FUNCTION_BLOCK fbDataExchangePIM
VAR_IN_OUT
	stMachineDataPIM : stPimMachineData;
END_VAR
VAR_INPUT
	//All purpose data
	sIpAdress 						: STRING(15);				// Ip Adress of machine
	iPort							: UINT;						// Port of the machine
	iUnitId							: BYTE;						// Id of Slave
	tCommunicationTimeOut			: TIME;						// Time until error 
	iCommunicationPerformEvery		: INT;						// Perform data exchange every ms
	bEnableCommunication			: BOOL;						// Enable communication
	//Byte purpose data
	wRegistersReadQuantity			: WORD;						// Amount of data do read
	wRegistersWriteQuantity			: WORD;						// Amount of data do read
	iRegisterReadStartAdress		: UINT;						// First adress of read registers data
	iRegisterWriteStartAdress		: UINT;						// First adress of write registers data
	iMaxCommunicationCycleTime		: INT;						//Maximum cycles to perform communication without error
END_VAR
VAR_OUTPUT
	bCommunicationError				: BOOL;						//Block state informaing about communication error
	iCommunicationErrorCode			: UDINT;					//Block state informaing about communication error
	bCommunicationBlockCycleExtended: BOOL;						//Communication Cycle extened
	iCommunicationCycleTime			: INT;						//
END_VAR

VAR
	iCommunicationStep 				: INT;	
	iCycleCalc						: INT;
	iLastCycleTimeClear				: TON;
	fbModbusTCP 					: FB_MBReadWriteRegs;
	arRegisterReadArray				: ARRAY[0..29] OF INT;
	arRegisterWriteArray			: ARRAY[0..29] OF INT;
	iHistoryError					: INT;
	arModbusErrorHist				: ARRAY[0..100] OF UDINT;
	iLasthistory					: INT;
END_VAR

//--------------------------------------------------------------------------------------------------
//Communication monitor
IF iCycleCalc > iMaxCommunicationCycleTime THEN
	bCommunicationError := TRUE;
	bCommunicationBlockCycleExtended := TRUE;
ELSIF fbModbusTCP.bError THEN
	bCommunicationError := TRUE;
	bCommunicationBlockCycleExtended := FALSE;
ELSE
	bCommunicationError := FALSE;
	bCommunicationBlockCycleExtended := FALSE;
END_IF
iCommunicationErrorCode := fbModbusTCP.nErrId;
IF iCycleCalc > iCommunicationCycleTime	  THEN
	iCommunicationCycleTime	:= iCycleCalc;
END_IF
iLastCycleTimeClear(IN:=TRUE,PT:=T#100MS);
IF iLastCycleTimeClear.Q THEN
	iCommunicationCycleTime := 0;
	iLastCycleTimeClear(IN:=FALSE);
END_IF
//--------------------------------------------------------------------------------------------------
//Statistic
//--------------------------------------------------------------------------------------------------
//Cycle counter
IF bEnableCommunication THEN
	iCycleCalc := iCycleCalc +1;
ELSE
	iCycleCalc := 0;
END_IF

//--------------------------------------------------------------------------------------------------
//SetUp for Ip Adress
fbModbusTCP.sIPAddr 			:= sIpAdress;
//--------------------------------------------------------------------------------------------------
//SetUp for Port No.
fbModbusTCP.nTCPPort 			:= iPort;
//--------------------------------------------------------------------------------------------------
//SetUp for Unit Id
fbModbusTCP.nUnitID 			:= iUnitId;
//--------------------------------------------------------------------------------------------------
//SetUp for TimeOut
fbModbusTCP.tTimeout 			:= tCommunicationTimeOut;
//--------------------------------------------------------------------------------------------------
//SetUp for First register
	//Read
fbModbusTCP.nMBReadAddr 		:= iRegisterReadStartAdress;
	//Write
fbModbusTCP.nMBWriteAddr 		:= iRegisterWriteStartAdress;
//--------------------------------------------------------------------------------------------------
//SetUp for data quantity
	//Read
fbModbusTCP.nReadQuantity 		:= UINT_TO_WORD(wRegistersReadQuantity);
	//Write
fbModbusTCP.nWriteQuantity 		:= UINT_TO_WORD(wRegistersWriteQuantity);
//--------------------------------------------------------------------------------------------------
//SetUp for data length
	//Read
fbModbusTCP.cbDestLength 		:= SIZEOF(arRegisterReadArray);
	//Write
fbModbusTCP.cbSrcLength 		:= SIZEOF(arRegisterWriteArray);
//--------------------------------------------------------------------------------------------------
//SetUp for data write adress
fbModbusTCP.pSrcAddr 			:= ADR(arRegisterWriteArray);
//--------------------------------------------------------------------------------------------------
//SetUp for data write adress
fbModbusTCP.pDestAddr 			:= ADR(arRegisterReadArray);

	//--------------------------------------------------------------------------------------------------
	//Background Operations
	fbModbusTCP();
	//--------------------------------------------------------------------------------------------------
	// Main loop for communication exchange
IF bEnableCommunication THEN
	CASE iCommunicationStep  OF 
		0:		//Initialization
		IF iCommunicationPerformEvery <= iCycleCalc THEN
			iCommunicationStep := 2;
			iCycleCalc := 0;
		END_IF
		2:		//Data setup
			//--------------------------------------------------------------------------------------------------
			// Data Write
			arRegisterWriteArray[0]					:= stMachineDataPIM.iProductId;
			arRegisterWriteArray[10]				:= BOOL_TO_INT(stMachineDataPIM.bLifeBitPLC);
			arRegisterWriteArray[11]				:= BOOL_TO_INT(stMachineDataPIM.bWorkAllow);
			arRegisterWriteArray[12]				:= BOOL_TO_INT(stMachineDataPIM.bResetError);
			arRegisterWriteArray[13]				:= BOOL_TO_INT(stMachineDataPIM.bConfirmError);
			arRegisterWriteArray[14]				:= BOOL_TO_INT(stMachineDataPIM.bTestMode);
			arRegisterWriteArray[15]				:= BOOL_TO_INT(stMachineDataPIM.bStopPerform);
			arRegisterWriteArray[18]				:= BOOL_TO_INT(stMachineDataPIM.bWaitWithWork);
			arRegisterWriteArray[19]				:= BOOL_TO_INT(stMachineDataPIM.bOfflineWorkAllow);
			iCommunicationStep := 5;
		5: 		//Read Coils
			//--------------------------------------------------------------------------------------------------
			// Perform data exchange
			fbModbusTCP.bExecute := TRUE;
			IF fbModbusTCP.bBusy THEN
				iCommunicationStep := 6;
				fbModbusTCP.bExecute := FALSE;
			END_IF
		6:		//Wait for end of 
			//--------------------------------------------------------------------------------------------------
			// Wait for end
			IF  NOT fbModbusTCP.bBusy THEN
				iCommunicationStep := 10;
			END_IF
		10:		//Read data form buffer
			//--------------------------------------------------------------------------------------------------
			// Data rewrite
			stMachineDataPIM.iActualWorkStep		:= arRegisterReadArray[0];
			stMachineDataPIM.wGoodPartsAmount		:= INT_TO_WORD(arRegisterReadArray[1]*256+arRegisterReadArray[2]);
			stMachineDataPIM.wBadPartsAmount		:= INT_TO_WORD(arRegisterReadArray[3]*256+arRegisterReadArray[4]);
			stMachineDataPIM.iCycleTime				:= arRegisterReadArray[5];
			stMachineDataPIM.iPartsCreatedInOneTime	:= arRegisterReadArray[6];
			stMachineDataPIM.iErrorCode				:= arRegisterReadArray[7];
			stMachineDataPIM.bLifeBitMachine		:= INT_TO_BOOL(arRegisterReadArray[10]);
			stMachineDataPIM.bWorkInProgress		:= INT_TO_BOOL(arRegisterReadArray[11]);
			stMachineDataPIM.bCycleEnd				:= INT_TO_BOOL(arRegisterReadArray[12]);
			stMachineDataPIM.bError					:= INT_TO_BOOL(arRegisterReadArray[13]);
			stMachineDataPIM.bAlarm					:= INT_TO_BOOL(arRegisterReadArray[14]);	
			//stMachineDataPIM.bOfflineWorkAllow		:= INT_TO_BOOL(arRegisterReadArray[15]);
			iCommunicationStep := 0;
	END_CASE
END_IF



IF fbModbusTCP.nErrId <> 0 AND iHistoryError > iLastHistory THEN
arModbusErrorHist[iHistoryError] := fbModbusTCP.nErrId;
iLasthistory := iHistoryError;
iHistoryError := iHistoryError + 1;
IF iHistoryError >= 100 THEN
	iHistoryError := 0;
	MEMSET(destAddr:=ADR(arModbusErrorHist),fillByte:=0,n:=SIZEOF(arModbusErrorHist));
END_IF
END_IF

END_FUNCTION_BLOCK

(* stored: Version 1.1.0.1, ProductVersion 3.1.4024.13
   POU fbDataExchangePIM: Id {e8ab9f09-9970-43bf-ae07-dd800a2d1129}, SpecialFunc None *)
